FUNCTION_BLOCK FIELDBUS_LINT_TO_SIGNAL (* Mirrors IN->OUT if Signal Valid. *)
  (* Standard: 61499-1 *)
  (* Version 1.0, 2026-05-31, franz *)
  PACKAGE logiBUS::signalprocessing::fieldbus;
  IMPORT signalprocessing::FIELDBUS_SIGNAL::NOT_AVAILABLE_DM;
  IMPORT signalprocessing::FIELDBUS_SIGNAL::VALID_SIGNAL_DW;
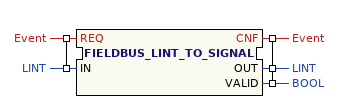
  EVENT_INPUT
    REQ WITH IN; (* Normal Execution Request *)
  END_EVENT
  EVENT_OUTPUT
    CNF WITH OUT, VALID; (* Execution Confirmation *)
  END_EVENT
  VAR_INPUT
    IN : LINT := DWORD_TO_LINT(NOT_AVAILABLE_DM); (* Input *)
  END_VAR
  VAR_OUTPUT
    OUT : LINT := 16#0000000000000000; (* Output Filtered *)
    VALID : BOOL := FALSE; (* TRUE if Signal is VALID *)
  END_VAR
  EC_STATES
    REQ : REQ -> CNF;
  END_STATES
  ALGORITHM REQ IN ST: (* Executed algorithm *)
IF (IN <= DWORD_TO_LINT(VALID_SIGNAL_DW)) THEN
	OUT := IN;
	VALID := BOOL#TRUE;
ELSE
	OUT := LINT#0;
	VALID := BOOL#FALSE;
END_IF;
  END_ALGORITHM
END_FUNCTION_BLOCK
